// SIMATIC S7-200 project (STEP 7-Micro/WIN), CPU 226 REL 02.01

ORGANIZATION_BLOCK 主程序:OB1
TITLE=程序注释
BEGIN
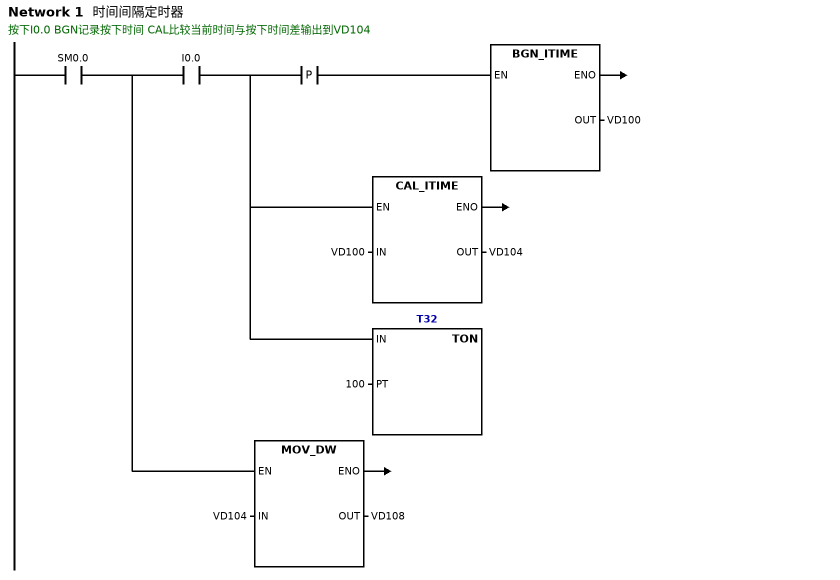
Network 1 // 时间间隔定时器
// 按下I0.0 BGN记录按下时间 CAL比较当前时间与按下时间差输出到VD104
LD     SM0.0
LPS
A      I0.0
LPS
EU
BITIM  VD100
LRD
CITIM  VD100, VD104
LPP
TON    T32, 100
LPP
MOVD   VD104, VD108
END_ORGANIZATION_BLOCK
